(* Logix 5000 project; controller test2 1756-L63 rev 19.15; software revision 19.01 *)

TASK MainTask (continuous, watchdog 500 ms) : MainProgram

MODULES
   Local : 1756-L63 (ICP 0, rev 19.15)
END_MODULES

ADD_ON_INSTRUCTION Motor   (* revision 1.2, vendor Kymera Systems Inc. *)
// Revision note:
// Update tag access
// Help:
// Motor Control Logic for both reversible and not-reversible motors
VAR_IN_OUT
   FirstOut : STRING; {required}   // First Out Interlock Text
END_VAR
VAR_INPUT
   IOValid : BOOL; {access Read Only}   // I/O Validation
   OperProgReq : BOOL;   // Boolean input to request a change to program mode from operator
   OperOperReq : BOOL;   // Boolean input to request a change to operator mode from operator
   OperOffReq : BOOL;   // Boolean input to request a change to OFF mode from operator
   OperMaintReq : BOOL;   // Boolean input to request a change to maintenance mode from operator
   ProgProgReq : BOOL;   // Boolean input to request a change to auto program mode
   ProgOperReq : BOOL;   // Boolean input to request a change to manual program mode
   ProgOffReq : BOOL;   // Program internal request to go in OFF mode
   OperStartReq : BOOL;   // Request by operator in Operator mode to Start the Motor
   OperStartReqRev : BOOL;   // Request by operator in Operator mode to Start the Motor in Reverse
   OperStopReq : BOOL;   // Request by operator in Operator mode to Stop the Motor
   ProgStartReq : BOOL;   // Request by Program in Program mode to Start the Motor
   ProgStopReq : BOOL;   // Request by Program in Program mode to Stop the Motor
   ProgStartReqRev : BOOL;   // Request by Program in Program mode to Start the Motor in Reverse
   ProgStopReqRev : BOOL;   // Request by Program in Program mode to Stop the Motor in Reverse
   GroupStartReq : BOOL;   // Group Request to Start the Motor
   GroupStartReqRev : BOOL;   // Group Request to Start the Motor in Reverse
   GroupStopReq : BOOL;   // Group Request to Stop the Motor
   IntkInitial : BOOL; {access Read Only, visible}   // Initial Interlock for Motor (Forward)
   IntkProcess : BOOL; {access Read Only, visible}   // Process Interlock for Motor (Forward)
   IntkSafety : BOOL; {access Read Only, visible}   // Safety Interlock for Motor (Forward)
   IntkMachine : BOOL; {access Read Only, visible}   // Machine Interlock for Motor (Forward)
   IntkInitialRev : BOOL; {access Read Only}   // Initial Interlock for Motor (Reverse)
   IntkProcessRev : BOOL; {access Read Only}   // Process Interlock for Motor (Reverse)
   IntkMachineRev : BOOL; {access Read Only}   // Machine Interlock for Motor (Reverse)
   IntkSafetyRev : BOOL; {access Read Only}   // Safety Interlock for Motor (Reverse)
   ExtTrip : BOOL; {access Read Only}   // External Trips input
   ManSpeedSP : REAL;   // Manual Speed SetPoint
   AutoSpeedSP : REAL;   // Auto Speed SetPoint
   MaxSpeedSP : REAL;   // Maximum Speed SetPoint
   MinSpeedSP : REAL;   // Minimum Speed SetPoint
   LocStart : BOOL; {access Read Only, visible}   // Local Start Command (Forward) (1 = ON)
   LocJog : BOOL; {access Read Only}   // Local Jog Command (Forward) (1 = ON)
   LocStartRev : BOOL; {access Read Only}   // Local Start Command (Reverse) (1 = ON)
   LocJogRev : BOOL; {access Read Only}   // Local Jog Command (Reverse) (1 = ON)
   LocStop : BOOL; {access Read Only, visible}   // Local Stop Command (0 = Stop)
   Overload : BOOL; {access Read Only}   // Overload Status (0 = TRIPPED)
   CPwr : BOOL; {access Read Only}   // Control Power Status (0 = TRIPPED)
   RunningFdbk : BOOL; {access Read Only, visible}   // Motor Running Feedback (Forward) (1 = Running)
   RunningFdbkRev : BOOL; {access Read Only}   // Motor Running Feedback (Reverse) (1 = Running)
   RemoteConnected : BOOL;   // Is the local HOA control switch used. True if Connected, False if else
   RemoteState : BOOL; {access Read Only}   // The status of the local HOA control switch. True if in Auto, False if else
   EStopConnected : BOOL;   // Is the Emergency Stop Push Button used. True if Connected, False if else
   EStop : BOOL; {access Read Only}   // Emergency Stop Push Button Status (0 = Stop)
   BellTime : DINT;   // The Time in which the Bell will be Ringing Before Starting the Motor
   FailStartTime : DINT;   // The Maximum Allowable Time Between the Start Command Change and the Running Feedback Activation (Forward)
   FailStartTimeRev : DINT;   // The Maximum Allowable Time Between the Start Command Change and the Running Feedback Activation (Reverse)
   Ack : BOOL;   // Acknowledge Signal
END_VAR
VAR_OUTPUT
   StsExtTrip : BOOL; {access Read Only, visible}   // Status of External Trips
   StsOverload : BOOL; {access Read Only}   // Status of the Overload Trip
   StsCPwr : BOOL; {access Read Only}   // Status of the Control Power Trip
   StsEStop : BOOL; {access Read Only}   // Emergency Stop Activated
   StsAvailable : BOOL; {access Read Only, visible}   // Status Available for the Motor Command (Forward)
   StsAvailableRev : BOOL; {access Read Only, visible}   // Status Available for the Motor Command (Reverse)
   StsReady : BOOL; {access Read Only, visible}   // Status Ready for the Motor Command (Forward)
   StsReadyRev : BOOL; {access Read Only}   // Status Ready for the Motor Command (Reverse)
   StsProg : BOOL; {access Read Only, visible}   // Status Program of the Motor
   StsOper : BOOL; {access Read Only, visible}   // Status Operator of the Motor
   StsMaint : BOOL; {access Read Only, visible}   // Status Maintenance of the Motor
   SpeedSP : REAL; {access Read Only}   // The Speed SetPoint Output
   StartCmd : BOOL; {access Read Only, visible}   // Output to Start the Motor (Forward)
   StartCmdRev : BOOL; {access Read Only}   // Output to Start the Motor (Reverse)
   StopCmd : BOOL; {access Read Only, visible}   // Output to Stop the Motor (Forward)
   StopCmdRev : BOOL; {access Read Only}   // Output to Stop the Motor (Reverse)
   StsRun : BOOL; {access Read Only, visible}   // Status Running of the Motor (Forward)
   StsRunRev : BOOL; {access Read Only}   // Status Running of the Motor (Reverse)
   RunTime : DINT; {access Read Only, visible}   // The Runtime Counter of the Motor (Forward)
   RunTimeRev : DINT; {access Read Only}   // The Runtime Counter of the Motor (Reverse)
   StartCount : DINT; {access Read Only, visible}   // The Start Counter of the Motor (Forward)
   StartCountRev : DINT; {access Read Only}   // The Start Counter of the Motor (Reverse)
   BellCmd : BOOL; {access Read Only}   // Output to Activate the Bell
   FailedToStart : BOOL; {access Read Only}   // Signal Indicating that the Running Feedback was not Activated in the Allocated Time (Forward)
   FailedToStartRev : BOOL; {access Read Only}   // Signal Indicating that the Running Feedback was not Activated in the Allocated Time (Reverse)
END_VAR
VAR
   LocStartTimer : TIMER := (PRE := 500);   // Timer to Check if the Local Start Input is Genuine (Forward)
   LocStartReq : BOOL;   // Local Start Request (Forward)
   StsLocStop : BOOL;   // Local Stop Request
   LocStopTimer : TIMER := (PRE := 500);   // Timer to Check if the Local Stop Input is Genuine
   RTORunHours : TIMER;   // Timer to Calculate Motor Running Time (Forward)
   ResetRunTime : BOOL;   // Reset Motor Runtime (Forward)
   SC : COUNTER;   // Motor Start Counter (Forward)
   ResetSC : BOOL;   // Reset Start Count (Forward)
   FailStartTimer : TIMER; {access None}   // Time to Check if the Maximum Time to get the Running Feedback is Elapsed (Forward)
   Start : BOOL; {access None}   // Motor Start Internal Command (Forward)
   BellTimer : TIMER; {access None}   // Timer to Ring the Bell
   RemoteActive : BOOL; {access Read Only}   // Remote Active State
   TmrIntlkRev : TIMER := (PRE := 1000); {access None}   // Timer To Check if the Forward Start Command and Running Feedback are Deactivated for the Specified Period of Time
   TmrIntlkFwd : TIMER := (PRE := 1000); {access None}   // Timer To Check if the Reverse Start Command and Running Feedback are Deactivated for the Specified Period of Time
   StartRev : BOOL; {access None}   // Motor Start Internal Command (Reverse)
   LocStartReqRev : BOOL; {access None}   // Local Start Request (Reverse)
   FailStartTimerRev : TIMER; {access None}   // Time to Check if the Maximum Time to get the Running Feedback is Elapsed (Reverse)
   RTORunHoursRev : TIMER; {access None}   // Timer to Calculate Motor Running Time (Reverse)
   ResetRunTimeRev : BOOL; {access None}   // Timer to Check if the Local Start Input is Genuine (Reverse)
   SCRev : COUNTER; {access None}   // Motor Start Counter (Reverse)
   ResetSCRev : BOOL; {access None}   // Timer to Check if the Local Start Input is Genuine (Reverse)
   OneShotStop : BOOL; {access None}   // Local Stop Trigger
   OneShotStart : BOOL; {access None}   // Local Start Trigger
   LocStartTimerRev : TIMER := (PRE := 500); {access None}   // Timer to Check if the Local Start Input is Genuine (Reverse)
   LocStopIntrlkText : STRING := 'Local Stop Trip'; {access Read Only}   // Local Stop Interlock Text
   FailedToStartText : STRING := 'Failed to Start Trip'; {access Read Only}   // Failed to Start Interlock Text
   FailedToStartRevText : STRING := 'Failed to Start Reverse'; {access Read Only}   // Failed to Start in Reverse Interlock Text
   EStopIntrlkText : STRING := 'Emergency Stop Trip'; {access Read Only}   // Emergency Stop Interlock Text
   LastRunDir : BOOL; {access None}   // Last running direction (1=Fwd, 0=Rev)
   EmptyIntrlkText : STRING; {access None}   // Empty Interlock Text
   Description : STRING;   // The Motor Description
   OverloadIntrlkText : STRING := 'Overload Trip'; {access Read Only}   // Overload Interlock Text
   CPwrIntrlkText : STRING := 'Control Power Trip'; {access Read Only}   // Control Power Interlock Text
   IntkSafetyLatched : BOOL; {access Read Only}   // Safety Interlock for Motor (Forward) Latched Status
   IntkMachineLatched : BOOL; {access Read Only}   // Machine Interlock for Motor (Forward) Latched Status
   IntkSafetyRevLatched : BOOL; {access Read Only}   // Safety Interlock for Motor (Reverse) Latched Status
   IntkMachineRevLatched : BOOL; {access Read Only}   // Machine Interlock for Motor (Reverse) Latched Status
   OneShotProgStart : BOOL; {access None}
   OneShotProgStartRev : BOOL; {access None}
   StartReset : BOOL; {access None}
   StartRevReset : BOOL; {access None}
END_VAR

ROUTINE Logic   (* ladder *)
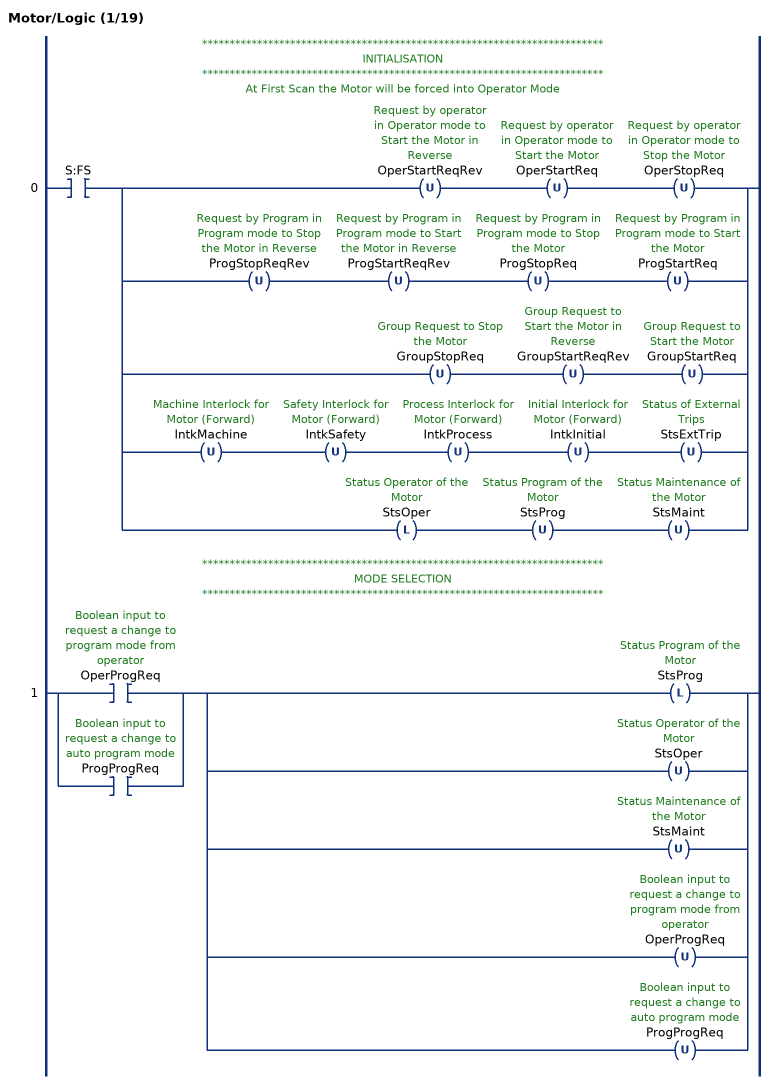
   // *************************************************************************
   // INITIALISATION
   // *************************************************************************
   // At First Scan the Motor will be forced into Operator Mode
   0: XIC(S:FS)[OTU(OperStartReqRev) OTU(OperStartReq) OTU(OperStopReq) ,OTU(ProgStopReqRev) OTU(ProgStartReqRev) OTU(ProgStopReq) OTU(ProgStartReq) ,OTU(GroupStopReq) OTU(GroupStartReqRev) OTU(GroupStartReq) ,OTU(IntkMachine) OTU(IntkSafety) OTU(IntkProcess) OTU(IntkInitial) OTU(StsExtTrip) ,OTL(StsOper) OTU(StsProg) OTU(StsMaint) ];
   // *************************************************************************
   // MODE SELECTION
   // *************************************************************************
   1: [XIC(OperProgReq) ,XIC(ProgProgReq) ][OTL(StsProg) ,OTU(StsOper) ,OTU(StsMaint) ,OTU(OperProgReq) ,OTU(ProgProgReq) ];
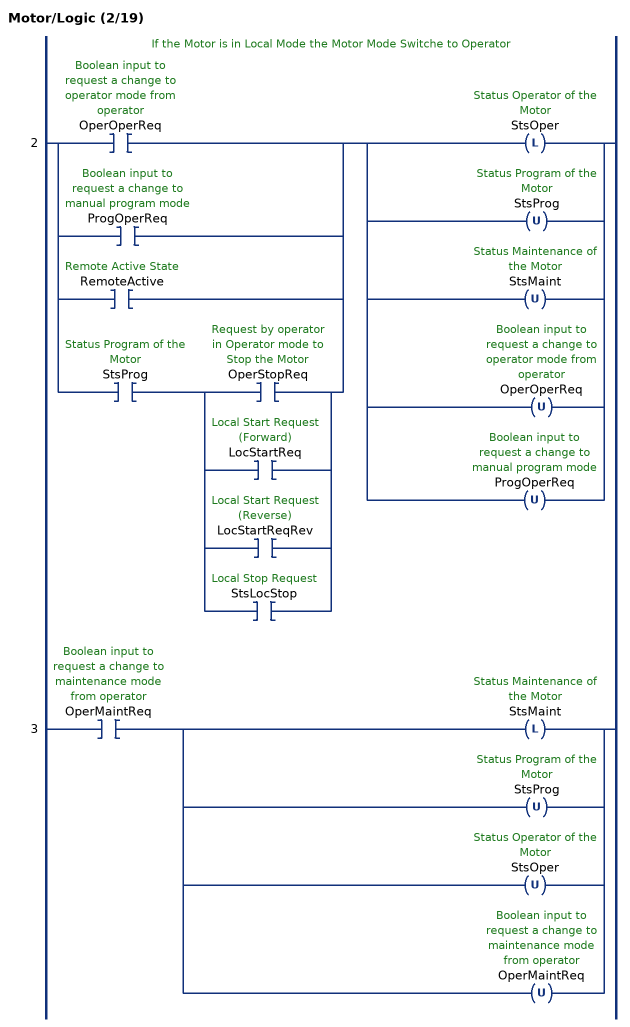
   // If the Motor is in Local Mode the Motor Mode Switche to Operator
   2: [XIC(OperOperReq) ,XIC(ProgOperReq) ,XIC(RemoteActive) ,XIC(StsProg) [XIC(OperStopReq) ,XIC(LocStartReq) ,XIC(LocStartReqRev) ,XIC(StsLocStop) ] ][OTL(StsOper) ,OTU(StsProg) ,OTU(StsMaint) ,OTU(OperOperReq) ,OTU(ProgOperReq) ];
   3: XIC(OperMaintReq)[OTL(StsMaint) ,OTU(StsProg) ,OTU(StsOper) ,OTU(OperMaintReq) ];
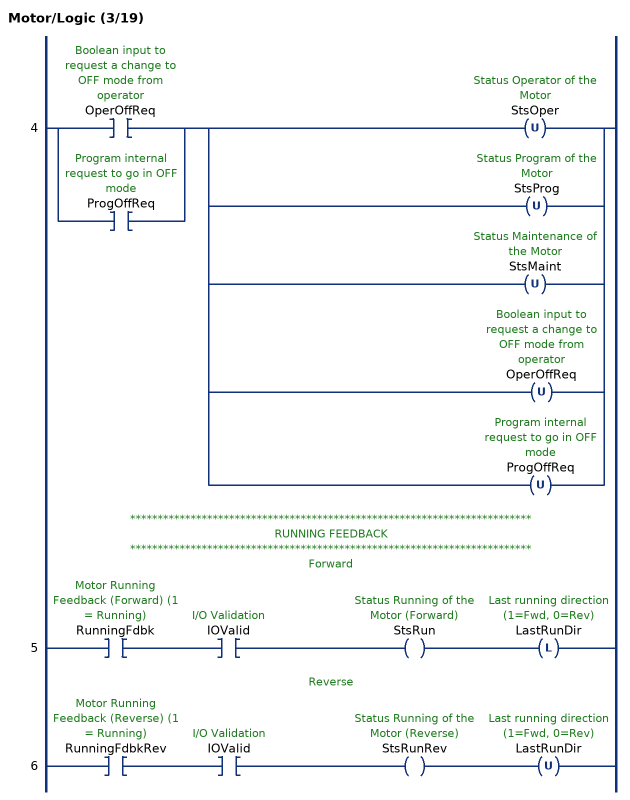
   4: [XIC(OperOffReq) ,XIC(ProgOffReq) ][OTU(StsOper) ,OTU(StsProg) ,OTU(StsMaint) ,OTU(OperOffReq) ,OTU(ProgOffReq) ];
   // *************************************************************************
   // RUNNING FEEDBACK
   // *************************************************************************
   // Forward
   5: XIC(RunningFdbk)XIC(IOValid)OTE(StsRun)OTL(LastRunDir);
   // Reverse
   6: XIC(RunningFdbkRev)XIC(IOValid)OTE(StsRunRev)OTU(LastRunDir);
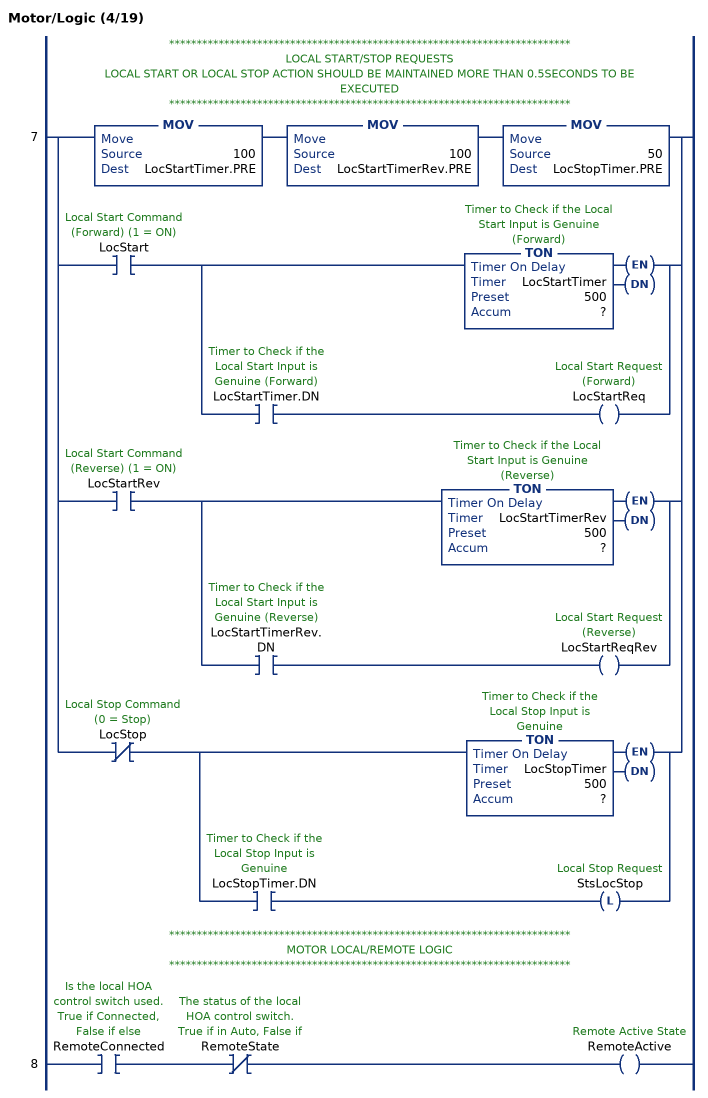
   // *************************************************************************
   // LOCAL START/STOP REQUESTS
   // LOCAL START OR LOCAL STOP ACTION SHOULD BE MAINTAINED MORE THAN 0.5SECONDS TO BE EXECUTED
   // *************************************************************************
   7: [MOV(100,LocStartTimer.PRE) MOV(100,LocStartTimerRev.PRE) MOV(50,LocStopTimer.PRE) ,XIC(LocStart) [TON(LocStartTimer,?,?) ,XIC(LocStartTimer.DN) OTE(LocStartReq) ] ,XIC(LocStartRev) [TON(LocStartTimerRev,?,?) ,XIC(LocStartTimerRev.DN) OTE(LocStartReqRev) ] ,XIO(LocStop) [TON(LocStopTimer,?,?) ,XIC(LocStopTimer.DN) OTL(StsLocStop) ] ];
   // *************************************************************************
   // MOTOR LOCAL/REMOTE LOGIC
   // *************************************************************************
   8: XIC(RemoteConnected)XIO(RemoteState)OTE(RemoteActive);
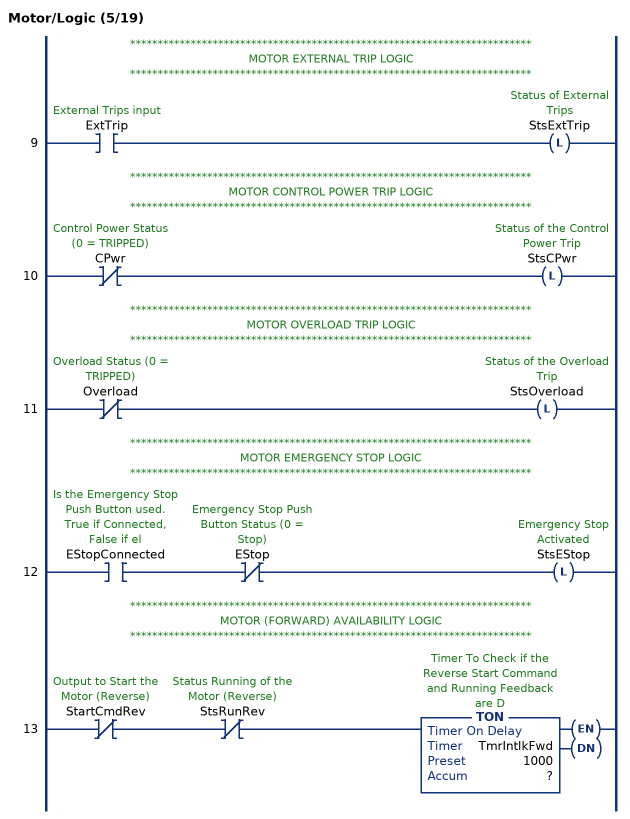
   // *************************************************************************
   // MOTOR EXTERNAL TRIP LOGIC
   // *************************************************************************
   9: XIC(ExtTrip)OTL(StsExtTrip);
   // *************************************************************************
   // MOTOR CONTROL POWER TRIP LOGIC
   // *************************************************************************
   10: XIO(CPwr)OTL(StsCPwr);
   // *************************************************************************
   // MOTOR OVERLOAD TRIP LOGIC
   // *************************************************************************
   11: XIO(Overload)OTL(StsOverload);
   // *************************************************************************
   // MOTOR EMERGENCY STOP LOGIC
   // *************************************************************************
   12: XIC(EStopConnected)XIO(EStop)OTL(StsEStop);
   // *************************************************************************
   // MOTOR (FORWARD) AVAILABILITY LOGIC
   // *************************************************************************
   13: XIO(StartCmdRev)XIO(StsRunRev)TON(TmrIntlkFwd,?,?);
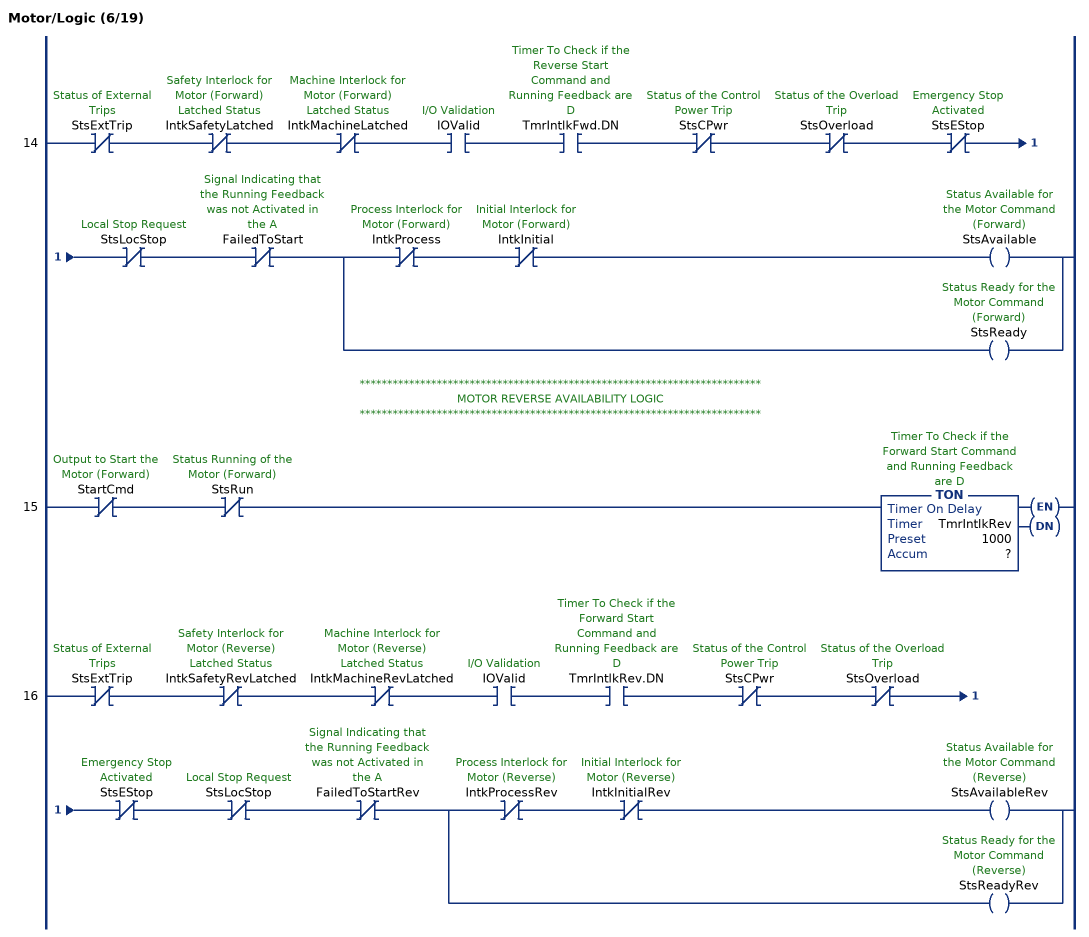
   14: XIO(StsExtTrip)XIO(IntkSafetyLatched)XIO(IntkMachineLatched)XIC(IOValid)XIC(TmrIntlkFwd.DN)XIO(StsCPwr)XIO(StsOverload)XIO(StsEStop)XIO(StsLocStop)XIO(FailedToStart)[XIO(IntkProcess) XIO(IntkInitial) OTE(StsAvailable) ,OTE(StsReady) ];
   // *************************************************************************
   // MOTOR REVERSE AVAILABILITY LOGIC
   // *************************************************************************
   15: XIO(StartCmd)XIO(StsRun)TON(TmrIntlkRev,?,?);
   16: XIO(StsExtTrip)XIO(IntkSafetyRevLatched)XIO(IntkMachineRevLatched)XIC(IOValid)XIC(TmrIntlkRev.DN)XIO(StsCPwr)XIO(StsOverload)XIO(StsEStop)XIO(StsLocStop)XIO(FailedToStartRev)[XIO(IntkProcessRev) XIO(IntkInitialRev) OTE(StsAvailableRev) ,OTE(StsReadyRev) ];
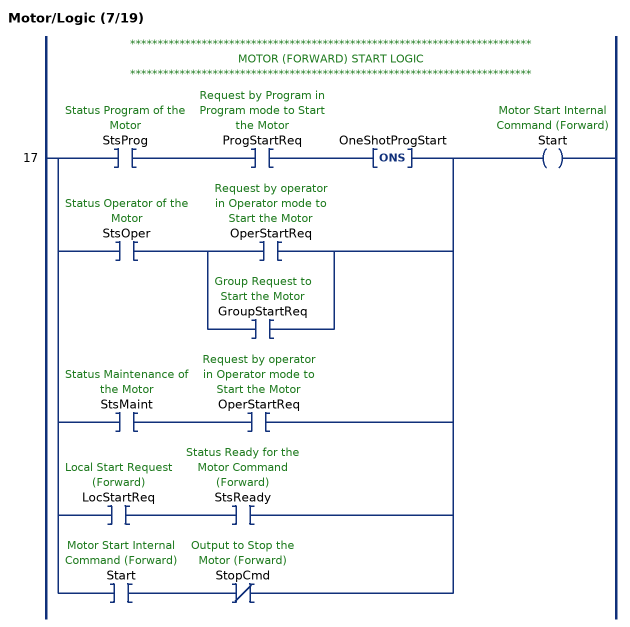
   // *************************************************************************
   // MOTOR (FORWARD) START LOGIC
   // *************************************************************************
   17: [XIC(StsProg) XIC(ProgStartReq) ONS(OneShotProgStart) ,XIC(StsOper) [XIC(OperStartReq) ,XIC(GroupStartReq) ] ,XIC(StsMaint) XIC(OperStartReq) ,XIC(LocStartReq) XIC(StsReady) ,XIC(Start) XIO(StopCmd) ]OTE(Start);
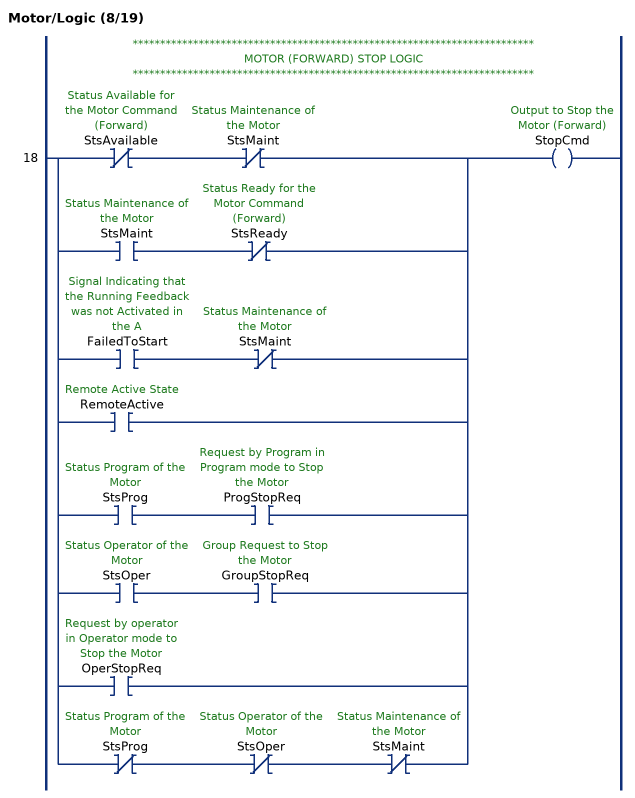
   // *************************************************************************
   // MOTOR (FORWARD) STOP LOGIC
   // *************************************************************************
   18: [XIO(StsAvailable) XIO(StsMaint) ,XIC(StsMaint) XIO(StsReady) ,XIC(FailedToStart) XIO(StsMaint) ,XIC(RemoteActive) ,XIC(StsProg) XIC(ProgStopReq) ,XIC(StsOper) XIC(GroupStopReq) ,XIC(OperStopReq) ,XIO(StsProg) XIO(StsOper) XIO(StsMaint) ]OTE(StopCmd);
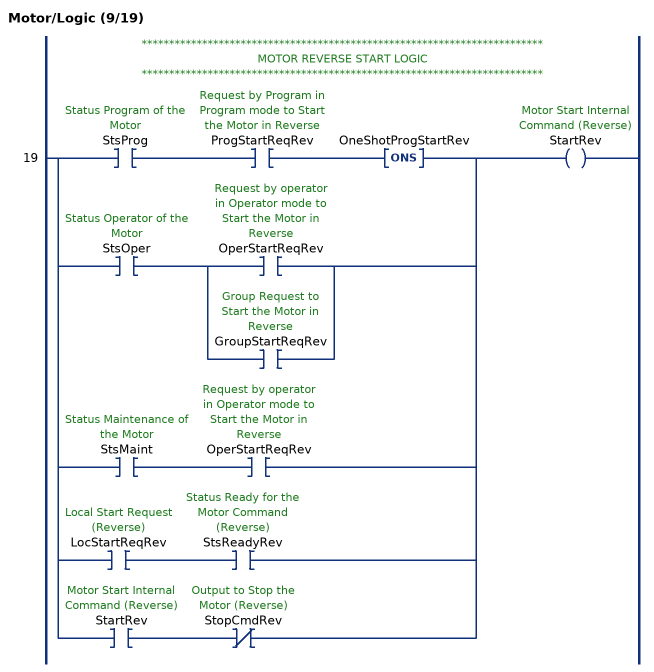
   // *************************************************************************
   // MOTOR REVERSE START LOGIC
   // *************************************************************************
   19: [XIC(StsProg) XIC(ProgStartReqRev) ONS(OneShotProgStartRev) ,XIC(StsOper) [XIC(OperStartReqRev) ,XIC(GroupStartReqRev) ] ,XIC(StsMaint) XIC(OperStartReqRev) ,XIC(LocStartReqRev) XIC(StsReadyRev) ,XIC(StartRev) XIO(StopCmdRev) ]OTE(StartRev);
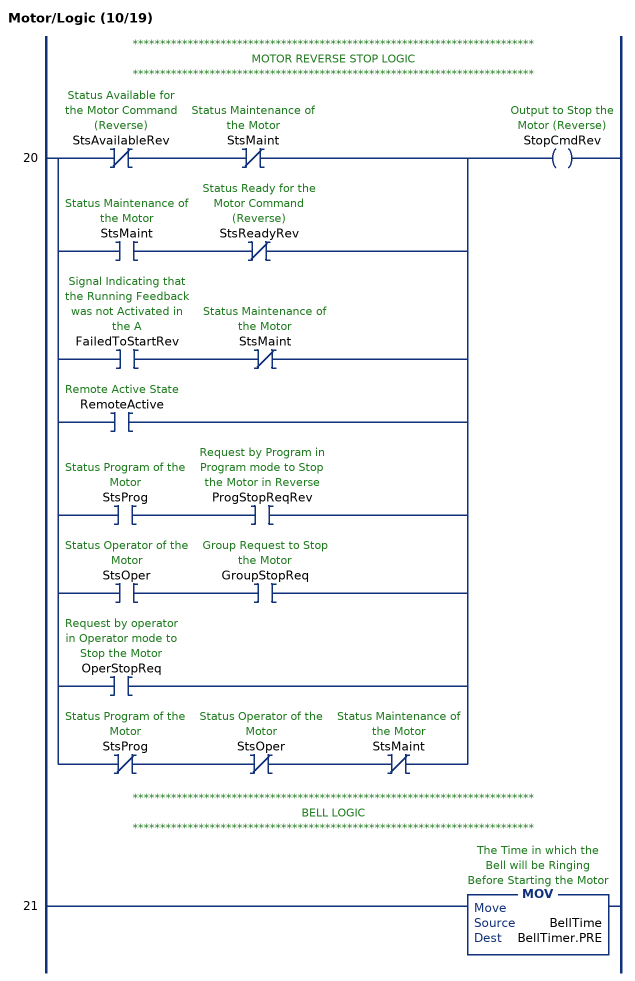
   // *************************************************************************
   // MOTOR REVERSE STOP LOGIC
   // *************************************************************************
   20: [XIO(StsAvailableRev) XIO(StsMaint) ,XIC(StsMaint) XIO(StsReadyRev) ,XIC(FailedToStartRev) XIO(StsMaint) ,XIC(RemoteActive) ,XIC(StsProg) XIC(ProgStopReqRev) ,XIC(StsOper) XIC(GroupStopReq) ,XIC(OperStopReq) ,XIO(StsProg) XIO(StsOper) XIO(StsMaint) ]OTE(StopCmdRev);
   // *************************************************************************
   // BELL LOGIC
   // *************************************************************************
   21: MOV(BellTime,BellTimer.PRE);
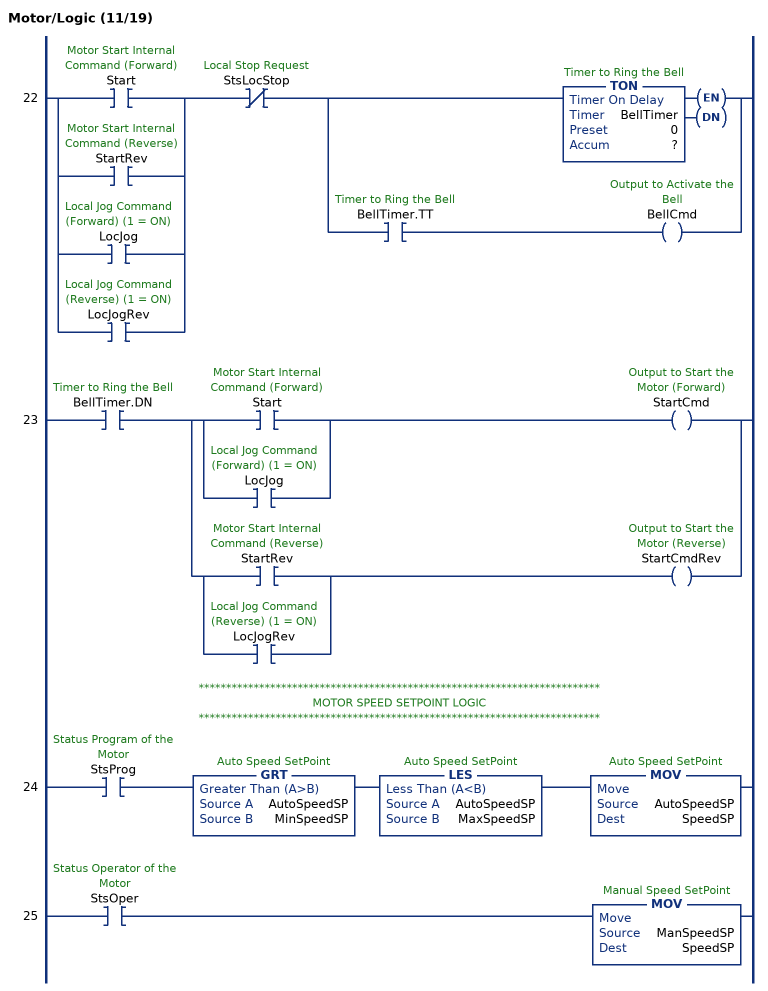
   22: [XIC(Start) ,XIC(StartRev) ,XIC(LocJog) ,XIC(LocJogRev) ]XIO(StsLocStop)[TON(BellTimer,?,?) ,XIC(BellTimer.TT) OTE(BellCmd) ];
   23: XIC(BellTimer.DN)[[XIC(Start) ,XIC(LocJog) ] OTE(StartCmd) ,[XIC(StartRev) ,XIC(LocJogRev) ] OTE(StartCmdRev) ];
   // *************************************************************************
   // MOTOR SPEED SETPOINT LOGIC
   // *************************************************************************
   24: XIC(StsProg)GRT(AutoSpeedSP,MinSpeedSP)LES(AutoSpeedSP,MaxSpeedSP)MOV(AutoSpeedSP,SpeedSP);
   25: XIC(StsOper)MOV(ManSpeedSP,SpeedSP);
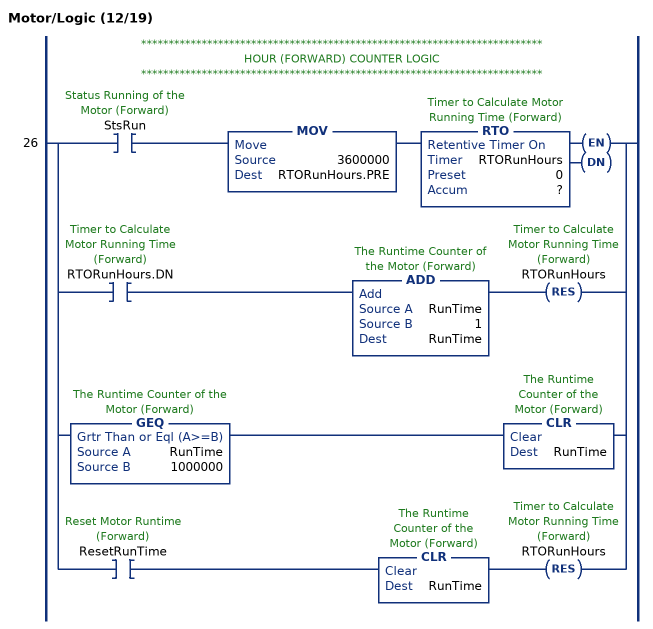
   // *************************************************************************
   // HOUR (FORWARD) COUNTER LOGIC
   // *************************************************************************
   26: [XIC(StsRun) MOV(3600000,RTORunHours.PRE) RTO(RTORunHours,?,?) ,XIC(RTORunHours.DN) ADD(RunTime,1,RunTime) RES(RTORunHours) ,GEQ(RunTime,1000000) CLR(RunTime) ,XIC(ResetRunTime) CLR(RunTime) RES(RTORunHours) ];
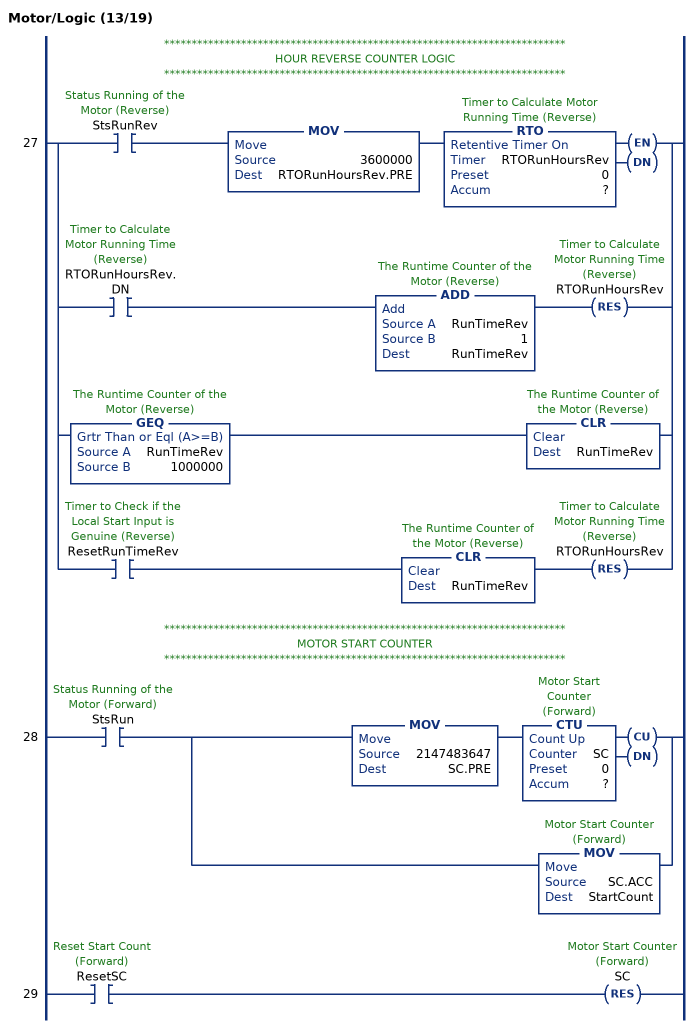
   // *************************************************************************
   // HOUR REVERSE COUNTER LOGIC
   // *************************************************************************
   27: [XIC(StsRunRev) MOV(3600000,RTORunHoursRev.PRE) RTO(RTORunHoursRev,?,?) ,XIC(RTORunHoursRev.DN) ADD(RunTimeRev,1,RunTimeRev) RES(RTORunHoursRev) ,GEQ(RunTimeRev,1000000) CLR(RunTimeRev) ,XIC(ResetRunTimeRev) CLR(RunTimeRev) RES(RTORunHoursRev) ];
   // *************************************************************************
   // MOTOR START COUNTER
   // *************************************************************************
   28: XIC(StsRun)[MOV(2147483647,SC.PRE) CTU(SC,?,?) ,MOV(SC.ACC,StartCount) ];
   29: XIC(ResetSC)RES(SC);
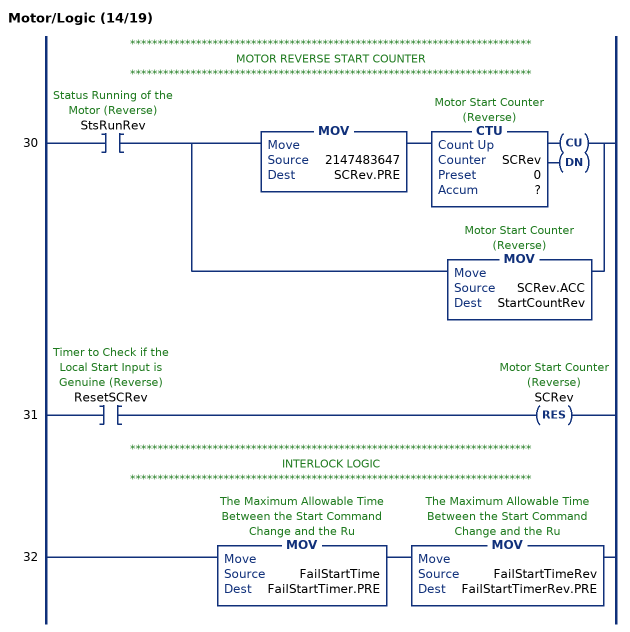
   // *************************************************************************
   // MOTOR REVERSE START COUNTER
   // *************************************************************************
   30: XIC(StsRunRev)[MOV(2147483647,SCRev.PRE) CTU(SCRev,?,?) ,MOV(SCRev.ACC,StartCountRev) ];
   31: XIC(ResetSCRev)RES(SCRev);
   // *************************************************************************
   // INTERLOCK LOGIC
   // *************************************************************************
   32: MOV(FailStartTime,FailStartTimer.PRE)MOV(FailStartTimeRev,FailStartTimerRev.PRE);
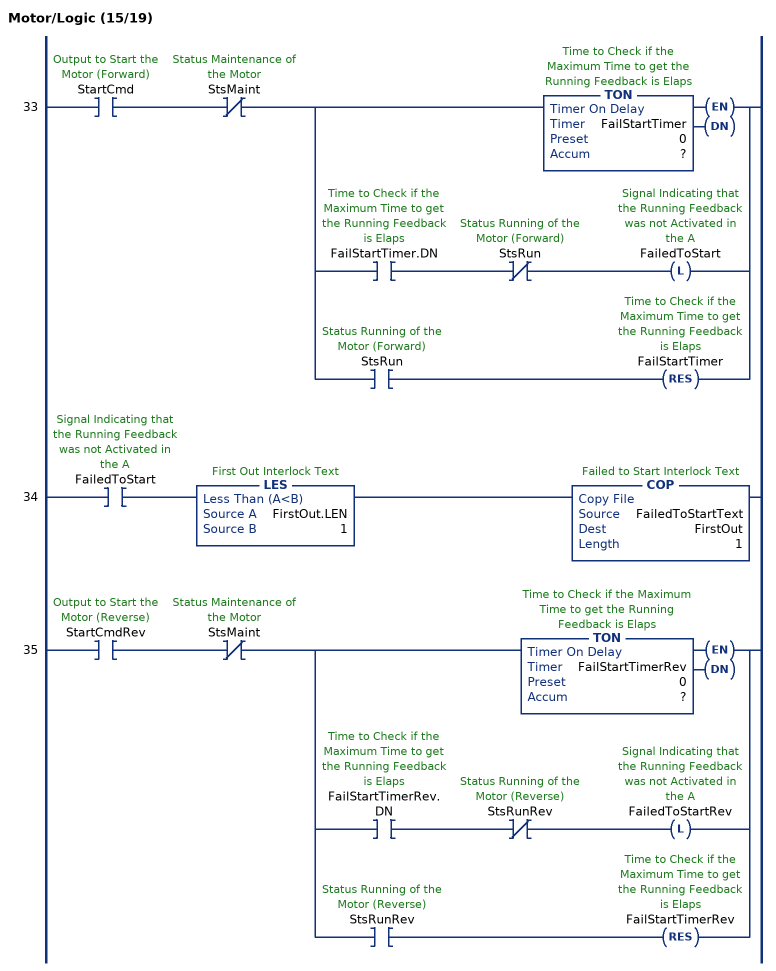
   33: XIC(StartCmd)XIO(StsMaint)[TON(FailStartTimer,?,?) ,XIC(FailStartTimer.DN) XIO(StsRun) OTL(FailedToStart) ,XIC(StsRun) RES(FailStartTimer) ];
   34: XIC(FailedToStart)LES(FirstOut.LEN,1)COP(FailedToStartText,FirstOut,1);
   35: XIC(StartCmdRev)XIO(StsMaint)[TON(FailStartTimerRev,?,?) ,XIC(FailStartTimerRev.DN) XIO(StsRunRev) OTL(FailedToStartRev) ,XIC(StsRunRev) RES(FailStartTimerRev) ];
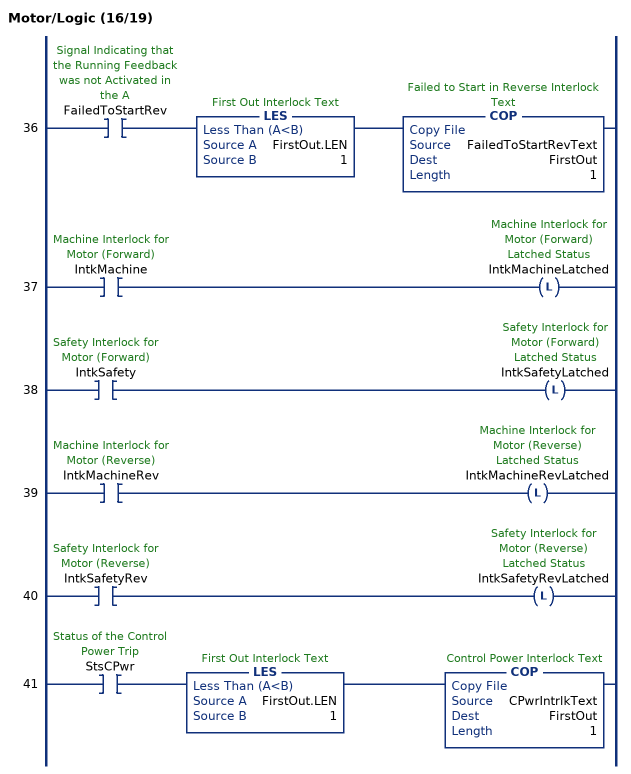
   36: XIC(FailedToStartRev)LES(FirstOut.LEN,1)COP(FailedToStartRevText,FirstOut,1);
   37: XIC(IntkMachine)OTL(IntkMachineLatched);
   38: XIC(IntkSafety)OTL(IntkSafetyLatched);
   39: XIC(IntkMachineRev)OTL(IntkMachineRevLatched);
   40: XIC(IntkSafetyRev)OTL(IntkSafetyRevLatched);
   41: XIC(StsCPwr)LES(FirstOut.LEN,1)COP(CPwrIntrlkText,FirstOut,1);
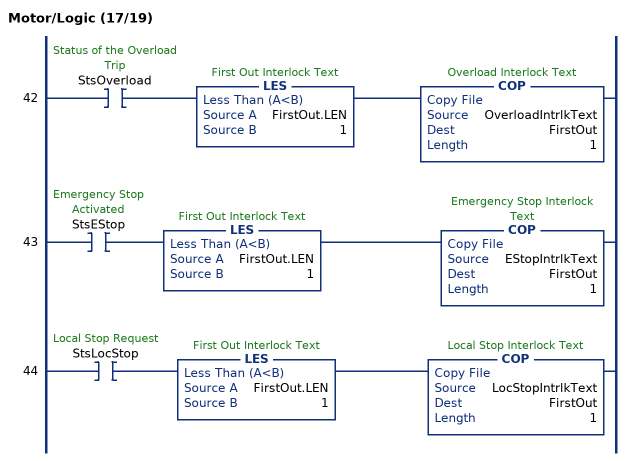
   42: XIC(StsOverload)LES(FirstOut.LEN,1)COP(OverloadIntrlkText,FirstOut,1);
   43: XIC(StsEStop)LES(FirstOut.LEN,1)COP(EStopIntrlkText,FirstOut,1);
   44: XIC(StsLocStop)LES(FirstOut.LEN,1)COP(LocStopIntrlkText,FirstOut,1);
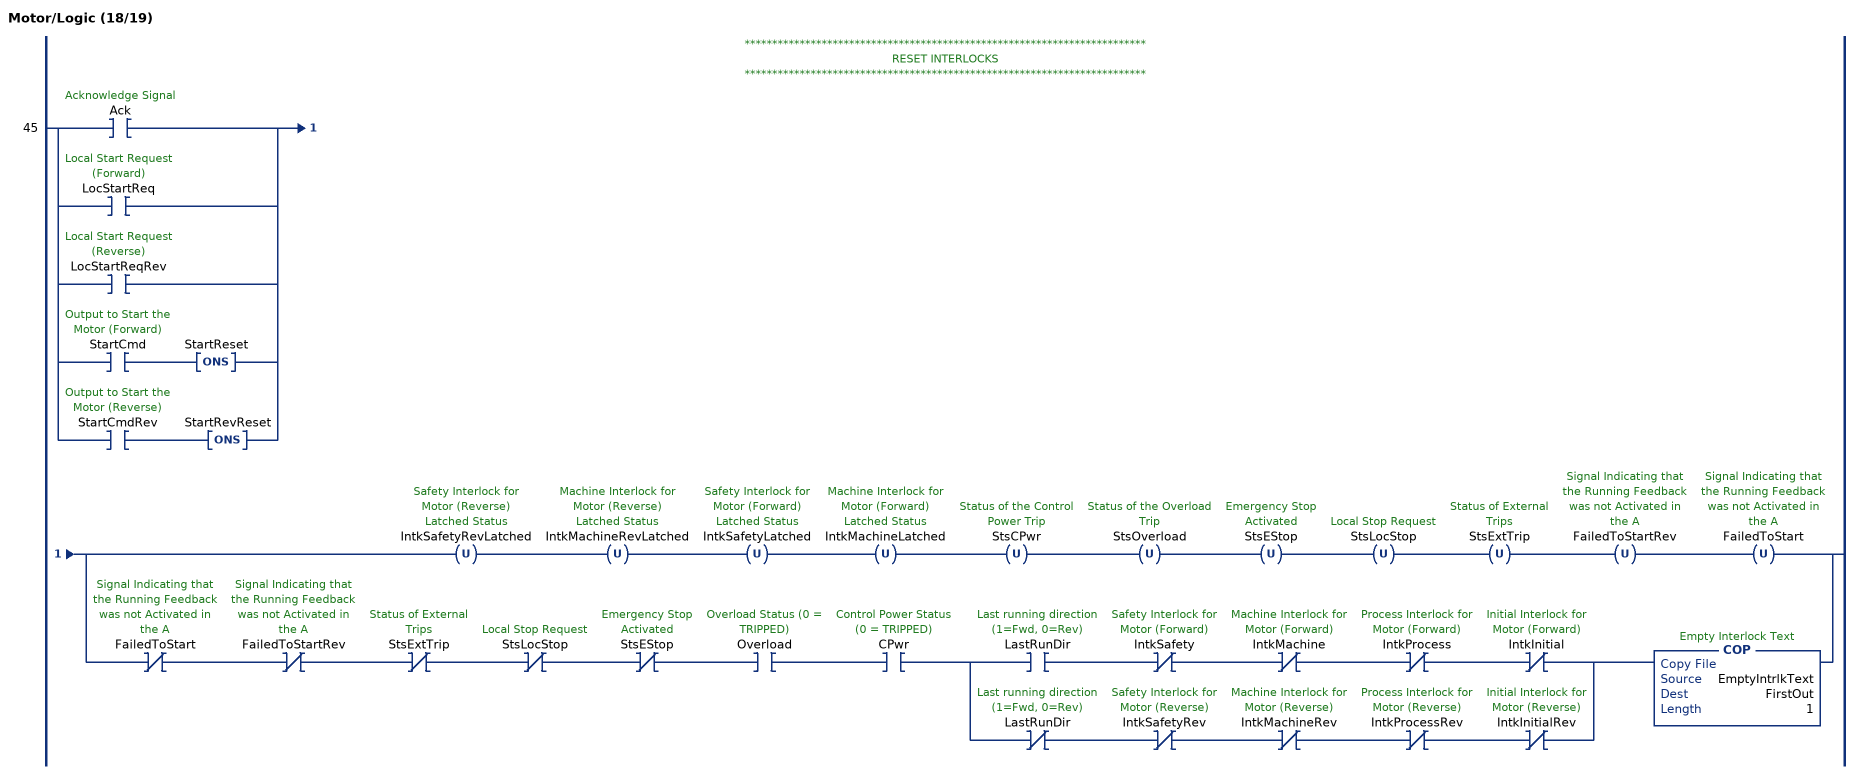
   // *************************************************************************
   // RESET INTERLOCKS
   // *************************************************************************
   45: [XIC(Ack) ,XIC(LocStartReq) ,XIC(LocStartReqRev) ,XIC(StartCmd) ONS(StartReset) ,XIC(StartCmdRev) ONS(StartRevReset) ][OTU(IntkSafetyRevLatched) OTU(IntkMachineRevLatched) OTU(IntkSafetyLatched) OTU(IntkMachineLatched) OTU(StsCPwr) OTU(StsOverload) OTU(StsEStop) OTU(StsLocStop) OTU(StsExtTrip) OTU(FailedToStartRev) OTU(FailedToStart) ,XIO(FailedToStart) XIO(FailedToStartRev) XIO(StsExtTrip) XIO(StsLocStop) XIO(StsEStop) XIC(Overload) XIC(CPwr) [XIC(LastRunDir) XIO(IntkSafety) XIO(IntkMachine) XIO(IntkProcess) XIO(IntkInitial) ,XIO(LastRunDir) XIO(IntkSafetyRev) XIO(IntkMachineRev) XIO(IntkProcessRev) XIO(IntkInitialRev) ] COP(EmptyIntrlkText,FirstOut,1) ];
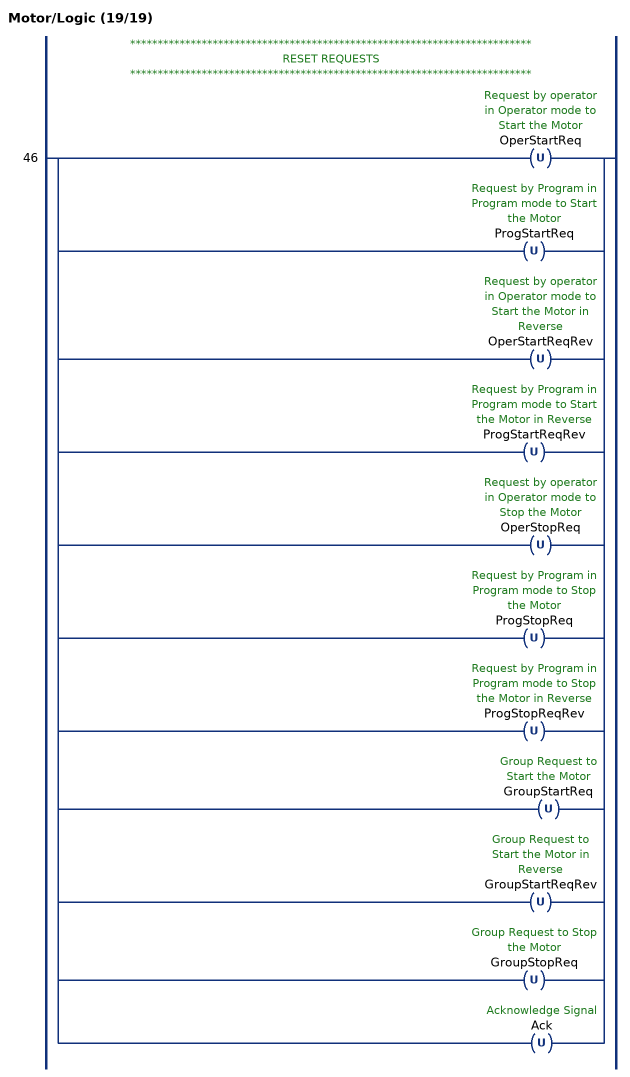
   // *************************************************************************
   // RESET REQUESTS
   // *************************************************************************
   46: [OTU(OperStartReq) ,OTU(ProgStartReq) ,OTU(OperStartReqRev) ,OTU(ProgStartReqRev) ,OTU(OperStopReq) ,OTU(ProgStopReq) ,OTU(ProgStopReqRev) ,OTU(GroupStartReq) ,OTU(GroupStartReqRev) ,OTU(GroupStopReq) ,OTU(Ack) ];
END_ROUTINE
END_ADD_ON_INSTRUCTION

PROGRAM MainProgram   (* main routine MainRoutine *)
VAR
   BillTimer : TIMER;
   C1 : COUNTER := (PRE := 10);
   Den_a : BOOL;
   Den_b : BOOL;
   Den_c : BOOL;
   Den_d : BOOL;
   FirstOut : STRING;
   IntkInitial : BOOL;
   IntkMachine : BOOL;
   IntkProcess : BOOL;
   IntkSafety : BOOL;
   LastRunDir : BOOL;
   LocStart : BOOL;
   LocStop : BOOL;
   Motor1 : Motor;
   OneShotProgStart : BOOL;
   Reset : BOOL;
   RunningFdbk : BOOL;
   RunTime : DINT;
   Start : BOOL := 1;
   StartCmd : BOOL;
   StartCount : DINT;
   StopCmd : BOOL;
   StsLocStart : BOOL;
   StsLocStop : BOOL;
   t1 : TIMER := (PRE := 1000);
   t2 : TIMER := (PRE := 2000);
END_VAR

ROUTINE MainRoutine   (* ladder *)
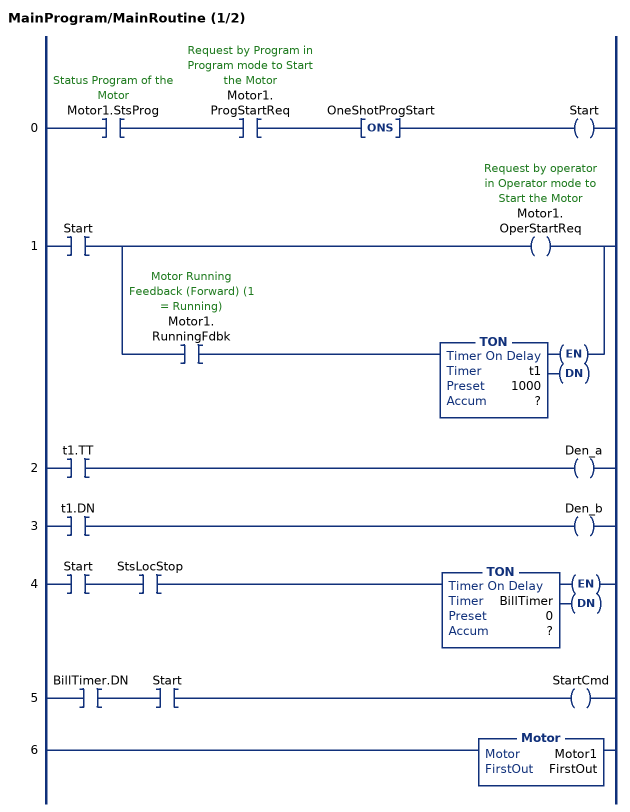
   0: XIC(Motor1.StsProg)XIC(Motor1.ProgStartReq)ONS(OneShotProgStart)OTE(Start);
   1: XIC(Start)[OTE(Motor1.OperStartReq) ,XIC(Motor1.RunningFdbk) TON(t1,?,?) ];
   2: XIC(t1.TT)OTE(Den_a);
   3: XIC(t1.DN)OTE(Den_b);
   4: XIC(Start)XIC(StsLocStop)TON(BillTimer,?,?);
   5: XIC(BillTimer.DN)XIC(Start)OTE(StartCmd);
   6: Motor(Motor1,FirstOut);
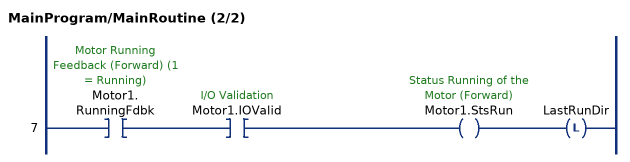
   7: XIC(Motor1.RunningFdbk)XIC(Motor1.IOValid)OTE(Motor1.StsRun)OTL(LastRunDir);
END_ROUTINE
END_PROGRAM
